% RSLogix 500 project I2P Hands On 1.RSS, saved by version 10.00.00.00 %
PROJECT "ML04A"    % processor: Bul.1763 MicroLogix 1100 Series B %

PROGRAM FILES
  LAD 2   5 rungs

DATA FILES
  O0 OUTPUT  4 elements
  I1 INPUT  6 elements
  S2 STATUS  66 elements
  B3 BINARY  1 elements
  T4 TIMER  1 elements
  C5 COUNTER  1 elements
  R6 CONTROL  1 elements
  N7 INTEGER  1 elements
  F8 FLOAT  1 elements

LADDER 2
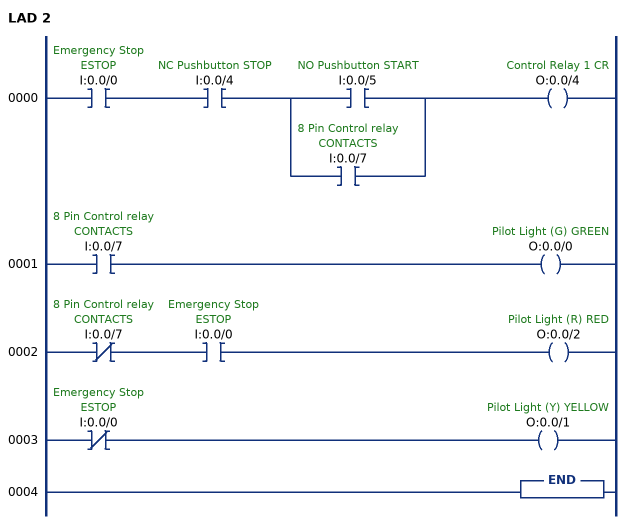
% Rung: 0 %
SOR XIC I:0.0/0 XIC I:0.0/4 BST XIC I:0.0/5 NXB XIC I:0.0/7 BND OTE O:0.0/4 EOR
%   I:0.0/0  ESTOP  "Emergency Stop" %
%   I:0.0/4  STOP  "NC Pushbutton" %
%   I:0.0/5  START  "NO Pushbutton" %
%   I:0.0/7  CONTACTS  "8 Pin Control relay" %
%   O:0.0/4  CR  "Control Relay 1" %
% Rung: 1 %
SOR XIC I:0.0/7 OTE O:0.0/0 EOR
%   I:0.0/7  CONTACTS  "8 Pin Control relay" %
%   O:0.0/0  GREEN  "Pilot Light (G)" %
% Rung: 2 %
SOR XIO I:0.0/7 XIC I:0.0/0 OTE O:0.0/2 EOR
%   I:0.0/7  CONTACTS  "8 Pin Control relay" %
%   I:0.0/0  ESTOP  "Emergency Stop" %
%   O:0.0/2  RED  "Pilot Light (R)" %
% Rung: 3 %
SOR XIO I:0.0/0 OTE O:0.0/1 EOR
%   I:0.0/0  ESTOP  "Emergency Stop" %
%   O:0.0/1  YELLOW  "Pilot Light (Y)" %
% Rung: 4 %
SOR END EOR

OTHER DOCUMENTED ADDRESSES
  I:0.0/1  FWD  "Three Position Selector Switch Position A"
  I:0.0/2  REV  "Three Position Selector Switch Position B"
  I:0.0/3  ON  "Two Position Selector Switch ON"
  I:0.0/6  JOG  "NO Pushbutton"
  O:0.0/3  BLUE  "Pilot Light (B)"
